(* IEC 61131-3 sources: com.logicals.lc3.webinar/usRTS_RPMControl_iSOC/src_FB_LIB_SAFE/Bitstring/LWORD, 10 files *)

(* ---- wAND_LWORD_2.iecst ---- *)
NAMESPACE logicals.web.standard
NAMESPACE bitstring

/*
 * Function block wrapper for IEC 61131-3 AND<br>
 * IN1 =  1st value (LWORD)<br>
 * IN2 =  2nd value (LWORD)<br>
 * OUT = IN1 AND IN2 (LWORD)<br>
 */
FUNCTION_BLOCK wAND_LWORD_2
	{ vNameAlignment:="center"; altName:="&"; bgColor:="DodgerBlue"; width:=40; hideIONames; }
	VAR_INPUT
		IN1 : LWORD;
		IN2 : LWORD;
	END_VAR
	VAR_OUTPUT
		OUT: LWORD;
	END_VAR

	OUT := AND(IN1:=IN1, IN2:=IN2, ENO=>ENO);
END_FUNCTION_BLOCK

END_NAMESPACE
END_NAMESPACE

(* ---- wAND_LWORD_3.iecst ---- *)
NAMESPACE logicals.web.standard
NAMESPACE bitstring

/*
 * Function block wrapper for IEC 61131-3 AND<br>
 * IN1 =  1st value (LWORD)<br>
 * IN2 =  2nd value (LWORD)<br>
 * IN3 =  3rd value (LWORD)<br>
 * OUT = IN1 AND IN2 AND IN3 (LWORD)<br>
 */
FUNCTION_BLOCK wAND_LWORD_3
	{ vNameAlignment:="center"; altName:="&"; bgColor:="DodgerBlue"; width:=40; hideIONames; }
	VAR_INPUT
		IN1 : LWORD;
		IN2 : LWORD;
		IN3 : LWORD;
	END_VAR
	VAR_OUTPUT
		OUT: LWORD;
	END_VAR

	OUT := AND(IN1:=IN1, IN2:=IN2, IN3:=IN3, ENO=>ENO);
END_FUNCTION_BLOCK

END_NAMESPACE
END_NAMESPACE

(* ---- wAND_LWORD_4.iecst ---- *)
NAMESPACE logicals.web.standard
NAMESPACE bitstring

/*
 * Function block wrapper for IEC 61131-3 AND<br>
 * IN1 =  1st value (LWORD)<br>
 * IN2 =  2nd value (LWORD)<br>
 * IN3 =  3rd value (LWORD)<br>
 * IN4 =  4th value (LWORD)<br>
 * OUT = IN1 AND IN2 AND IN3 AND IN4 (LWORD)<br>
 */
FUNCTION_BLOCK wAND_LWORD_4
	{ vNameAlignment:="center"; altName:="&"; bgColor:="DodgerBlue"; width:=40; hideIONames; }
	VAR_INPUT
		IN1 : LWORD;
		IN2 : LWORD;
		IN3 : LWORD;
		IN4 : LWORD;
	END_VAR
	VAR_OUTPUT
		OUT: LWORD;
	END_VAR

	OUT := AND(IN1:=IN1, IN2:=IN2, IN3:=IN3, IN4:=IN4, ENO=>ENO);
END_FUNCTION_BLOCK

END_NAMESPACE
END_NAMESPACE

(* ---- wNOT_LWORD.iecst ---- *)
NAMESPACE logicals.web.standard
NAMESPACE bitstring

/*
 * Function block wrapper for IEC 61131-3 NOT<br>
 * IN = input (LWORD)<br>
 * OUT = !IN (LWORD)<br>
 */
FUNCTION_BLOCK wNOT_LWORD
	{ vNameAlignment:="center"; altName:="NOT"; bgColor:="DodgerBlue"; width:=60; hideIONames; }
	VAR_INPUT
		IN : LWORD;
	END_VAR
	VAR_OUTPUT
		OUT: LWORD;
	END_VAR

	OUT := NOT(IN:=IN, ENO=>ENO);
END_FUNCTION_BLOCK

END_NAMESPACE
END_NAMESPACE

(* ---- wOR_LWORD_2.iecst ---- *)
NAMESPACE logicals.web.standard
NAMESPACE bitstring

/*
 * Function block wrapper for IEC 61131-3 OR<br>
 * IN1 =  1st value (LWORD)<br>
 * IN2 =  2nd value (LWORD)<br>
 * OUT = IN1 OR IN2 (LWORD)<br>
 */
FUNCTION_BLOCK wOR_LWORD_2
	{ vNameAlignment:="center"; altName:=">=1"; bgColor:="DodgerBlue"; width:=40; hideIONames; }
	VAR_INPUT
		IN1 : LWORD;
		IN2 : LWORD;
	END_VAR
	VAR_OUTPUT
		OUT: LWORD;
	END_VAR

	OUT := OR(IN1:=IN1, IN2:=IN2, ENO=>ENO);
END_FUNCTION_BLOCK

END_NAMESPACE
END_NAMESPACE

(* ---- wOR_LWORD_3.iecst ---- *)
NAMESPACE logicals.web.standard
NAMESPACE bitstring

/*
 * Function block wrapper for IEC 61131-3 OR<br>
 * IN1 =  1st value (LWORD)<br>
 * IN2 =  2nd value (LWORD)<br>
 * IN3 =  3rd value (LWORD)<br>
 * OUT = IN1 OR IN2 OR IN3 (LWORD)<br>
 */
FUNCTION_BLOCK wOR_LWORD_3
	{ vNameAlignment:="center"; altName:=">=1"; bgColor:="DodgerBlue"; width:=40; hideIONames; }
	VAR_INPUT
		IN1 : LWORD;
		IN2 : LWORD;
		IN3 : LWORD;
	END_VAR
	VAR_OUTPUT
		OUT: LWORD;
	END_VAR

	OUT := OR(IN1:=IN1, IN2:=IN2, IN3:=IN3, ENO=>ENO);
END_FUNCTION_BLOCK

END_NAMESPACE
END_NAMESPACE

(* ---- wOR_LWORD_4.iecst ---- *)
NAMESPACE logicals.web.standard
NAMESPACE bitstring

/*
 * Function block wrapper for IEC 61131-3 OR<br>
 * IN1 =  1st value (LWORD)<br>
 * IN2 =  2nd value (LWORD)<br>
 * IN3 =  3rd value (LWORD)<br>
 * IN4 =  4th value (LWORD)<br>
 * OUT = IN1 OR IN2 OR IN3 OR IN4 (LWORD)<br>
 */
FUNCTION_BLOCK wOR_LWORD_4
	{ vNameAlignment:="center"; altName:=">=1"; bgColor:="DodgerBlue"; width:=40; hideIONames; }
	VAR_INPUT
		IN1 : LWORD;
		IN2 : LWORD;
		IN3 : LWORD;
		IN4 : LWORD;
	END_VAR
	VAR_OUTPUT
		OUT: LWORD;
	END_VAR

	OUT := OR(IN1:=IN1, IN2:=IN2, IN3:=IN3, IN4:=IN4, ENO=>ENO);
END_FUNCTION_BLOCK

END_NAMESPACE
END_NAMESPACE

(* ---- wXOR_LWORD_2.iecst ---- *)
NAMESPACE logicals.web.standard
NAMESPACE bitstring

/*
 * Function block wrapper for IEC 61131-3 XOR<br>
 * IN1 =  1st value (LWORD)<br>
 * IN2 =  2nd value (LWORD)<br>
 * OUT = IN1 XOR IN2 (LWORD)<br>
 */
FUNCTION_BLOCK wXOR_LWORD_2
	{ vNameAlignment:="center"; altName:="=2k+1"; bgColor:="DodgerBlue"; width:=50; hideIONames; }
	VAR_INPUT
		IN1 : LWORD;
		IN2 : LWORD;
	END_VAR
	VAR_OUTPUT
		OUT: LWORD;
	END_VAR

	OUT := XOR(IN1:=IN1, IN2:=IN2, ENO=>ENO);
END_FUNCTION_BLOCK

END_NAMESPACE
END_NAMESPACE

(* ---- wXOR_LWORD_3.iecst ---- *)
NAMESPACE logicals.web.standard
NAMESPACE bitstring

/*
 * Function block wrapper for IEC 61131-3 XOR<br>
 * IN1 =  1st value (LWORD)<br>
 * IN2 =  2nd value (LWORD)<br>
 * IN3 =  3rd value (LWORD)<br>
 * OUT = IN1 XOR IN2 XOR IN3 (LWORD)<br>
 */
FUNCTION_BLOCK wXOR_LWORD_3
	{ vNameAlignment:="center"; altName:="=2k+1"; bgColor:="DodgerBlue"; width:=50; hideIONames; }
	VAR_INPUT
		IN1 : LWORD;
		IN2 : LWORD;
		IN3 : LWORD;
	END_VAR
	VAR_OUTPUT
		OUT: LWORD;
	END_VAR

	OUT := XOR(IN1:=IN1, IN2:=IN2, IN3:=IN3, ENO=>ENO);
END_FUNCTION_BLOCK

END_NAMESPACE
END_NAMESPACE

(* ---- wXOR_LWORD_4.iecst ---- *)
NAMESPACE logicals.web.standard
NAMESPACE bitstring

/*
 * Function block wrapper for IEC 61131-3 XOR<br>
 * IN1 =  1st value (LWORD)<br>
 * IN2 =  2nd value (LWORD)<br>
 * IN3 =  3rd value (LWORD)<br>
 * IN4 =  4th value (LWORD)<br>
 * OUT = IN1 XOR IN2 XOR IN3 XOR IN4 (LWORD)<br>
 */
FUNCTION_BLOCK wXOR_LWORD_4
	{ vNameAlignment:="center"; altName:="=2k+1"; bgColor:="DodgerBlue"; width:=50; hideIONames; }
	VAR_INPUT
		IN1 : LWORD;
		IN2 : LWORD;
		IN3 : LWORD;
		IN4 : LWORD;
	END_VAR
	VAR_OUTPUT
		OUT: LWORD;
	END_VAR

	OUT := XOR(IN1:=IN1, IN2:=IN2, IN3:=IN3, IN4:=IN4, ENO=>ENO);
END_FUNCTION_BLOCK

END_NAMESPACE
END_NAMESPACE
